FUNCTION_BLOCK AssemblyContainer EXTENDS ZCore.ObjectContainer
VAR_INPUT
END_VAR
VAR_OUTPUT
END_VAR
VAR
  {attribute 'hide'}
  _parent : REFERENCE TO AssemblyUnit;
END_VAR

{ attribute 'hide' }
METHOD FB_init : BOOL
VAR_INPUT
	bInitRetains : BOOL; // if TRUE, the retain variables are initialized (warm start / cold start)
	bInCopyCode : BOOL;  // if TRUE, the instance afterwards gets moved into the copy code (online change)
  unit : REFERENCE TO AssemblyUnit;
END_VAR
_parent REF= unit;
END_METHOD

END_FUNCTION_BLOCK

(* stored: Version 1.1.0.1
   POU AssemblyContainer: Id {5061d47b-591a-4b59-ae19-fc6bfe9e7cd6}, SpecialFunc None
   Method FB_init: Id {b8dbe970-4305-494d-a3f1-7747c9d0a4bc} *)
